END_FUNCTION_BLOCK

// ---- Observer Pattern/Abstraction/FB_AbstractObservable.TcPOU
FUNCTION_BLOCK ABSTRACT FB_AbstractObservable EXTENDS FB_Object IMPLEMENTS I_Observable
VAR
    // Attributes
    _nTypeClass:                __SYSTEM.TYPE_CLASS;
    _bAutoNotify:               BOOL := TRUE; // Notify automatically on write access of observable value
    _bNotifyWhenChanged:        BOOL; // Notify only when the value is actually changed

    // Dynamic mem
    _fbObsList:                 FB_List(0); // Observer list

    _fbNotifyObservers:         FB_NotifyObserverAction;
END_VAR

METHOD Attach : BOOL
VAR_INPUT
    ipObserver:     I_Observer;
END_VAR
IF ipObserver = 0 // Invalid interface pointer
    OR_ELSE ipObserver.nTypeClass <> THIS^._nTypeClass // Invalid type
    OR_ELSE THIS^.Contains(ipObserver) // Already added
    THEN
    RETURN;
END_IF

Attach := THIS^._fbObsList.AddItem(ipObserver) <> -1;

IF Attach THEN
    THIS^.NotifyLast();
END_IF
END_METHOD

(*Notify automatically on write access of observable value*)
PROPERTY bAutoNotify : BOOL
GET
bAutoNotify := THIS^._bAutoNotify;
END_GET
SET
THIS^._bAutoNotify := bAutoNotify;
END_SET
END_PROPERTY

PROPERTY bNotifyWhenChanged : BOOL
GET
bNotifyWhenChanged := THIS^._bNotifyWhenChanged;
END_GET
SET
THIS^._bNotifyWhenChanged := bNotifyWhenChanged;
END_SET
END_PROPERTY

METHOD ClearAll
VAR_INPUT
END_VAR
THIS^._fbObsList.Clear();
END_METHOD

METHOD Contains : BOOL
VAR_INPUT
    ipObserver: I_Observer;
END_VAR
Contains := THIS^._fbObsList.Contains(ipObserver);
END_METHOD

METHOD Detach : BOOL
VAR_INPUT
    ipObserver:     I_Observer;
END_VAR
Detach := THIS^._fbObsList.Remove(ipObserver);
END_METHOD

PROPERTY ABSTRACT nDataSize : UDINT
GET
END_GET
END_PROPERTY

PROPERTY nObserverCount : UDINT
GET
nObserverCount := THIS^._fbObsList.nCount;
END_GET
END_PROPERTY

METHOD NotifyAll : I_Observable
NotifyAll := THIS^;

THIS^._fbObsList.ForEach(
    THIS^._fbNotifyObservers
         .Inputs(THIS^.pData,
                 THIS^._nTypeClass,
                 THIS^.nDataSize));
END_METHOD

METHOD NotifyLast : I_Observable
VAR
    ipLastObs: I_Observer;
END_VAR
NotifyLast := THIS^;

ipLastObs := THIS^.ObserverAt(TO_DINT(THIS^.nObserverCount) - 1);

IF ipLastObs <> 0 THEN
    ipLastObs.UpdateP(pData := THIS^.pData,
                      nTypeClass := THIS^._nTypeClass,
                      nSize := THIS^.nDataSize);
END_IF
END_METHOD

METHOD PROTECTED NotifyWithConditions : I_Observable
VAR_INPUT
END_VAR
NotifyWithConditions := THIS^;

IF NOT THIS^._bAutoNotify THEN
    RETURN;
END_IF

IF THIS^._bNotifyWhenChanged
    AND_THEN NOT THIS^.ValueChanged() THEN
    RETURN;
END_IF

THIS^.NotifyAll();
END_METHOD

PROPERTY nTypeClass : __SYSTEM.TYPE_CLASS
GET
nTypeClass := THIS^._nTypeClass;
END_GET
END_PROPERTY

METHOD ObserverAt : I_Observer
VAR_INPUT
    nIdx: DINT;
END_VAR
__QUERYINTERFACE(THIS^._fbObsList.ItemAt(nIdx), ObserverAt);
END_METHOD

PROPERTY PROTECTED ABSTRACT pData : POINTER TO BYTE
GET
END_GET
END_PROPERTY

METHOD ABSTRACT ValueChanged : BOOL
VAR_INPUT
END_VAR
END_METHOD

END_FUNCTION_BLOCK

// ---- Observer Pattern/Abstraction/Actions/FB_NotifyObserverAction.TcPOU
FUNCTION_BLOCK FB_NotifyObserverAction EXTENDS FB_Action
VAR
    _pData: POINTER TO BYTE;
    _nSize: UDINT;
    _nTypeClass: __SYSTEM.TYPE_CLASS;
END_VAR

METHOD  Execute
VAR_INPUT
    ipObject: I_Object;
END_VAR
VAR
    ipObs: I_Observer;
END_VAR
__QUERYINTERFACE(ipObject, ipObs);

IF ipObs = 0 THEN
    RETURN;
END_IF

ipObs.UpdateP(pData := THIS^._pData,
              nTypeClass := THIS^._nTypeClass,
              nSize := THIS^._nSize);
END_METHOD

METHOD Inputs : I_Action
VAR_INPUT
    pData:          POINTER TO BYTE;
    nTypeClass:     __SYSTEM.TYPE_CLASS;
    nSize:          UDINT;
END_VAR
Inputs := THIS^;

THIS^._pData := pData;
THIS^._nTypeClass := nTypeClass;
THIS^._nSize := nSize;
END_METHOD

END_FUNCTION_BLOCK

// ---- Observer Pattern/FB_Observer_REAL.TcPOU
FUNCTION_BLOCK FB_Observer_REAL EXTENDS FB_AbstractObserver
VAR
    _fVal:              REAL;
END_VAR

METHOD FB_init : BOOL
VAR_INPUT
	bInitRetains : BOOL; // if TRUE, the retain variables are initialized (warm start / cold start)
	bInCopyCode : BOOL;  // if TRUE, the instance afterwards gets moved into the copy code (online change)
END_VAR
THIS^._nTypeClass := __SYSTEM.TYPE_CLASS.TYPE_REAL;
THIS^._pVal := ADR(THIS^._fVal);
THIS^._nSize := SIZEOF(THIS^._fVal);
END_METHOD

PROPERTY fValue32 : REAL
GET
fValue32 := THIS^._fVal;
END_GET
END_PROPERTY

END_FUNCTION_BLOCK

// ---- Observer Pattern/Abstraction/FB_AbstractObserver.TcPOU
FUNCTION_BLOCK ABSTRACT FB_AbstractObserver EXTENDS FB_Object IMPLEMENTS I_Observer
VAR
    _nTypeClass:        __SYSTEM.TYPE_CLASS;
    _pVal:              POINTER TO BYTE;
    _nSize:             DINT;
    _nUpdateCounter:    UDINT;
END_VAR

METHOD PROTECTED _Update
VAR_INPUT
    pData:          POINTER TO BYTE;
    nTypeClass:     __SYSTEM.TYPE_CLASS;
    nSize:          UDINT;
END_VAR
VAR
    nMemcpyRes:     UDINT;
END_VAR
IF nTypeClass <> THIS^._nTypeClass THEN
    RETURN;
END_IF

IF nSize <> TO_UDINT(THIS^._nSize) THEN
    RETURN;
END_IF

IF pData = 0 THEN
    RETURN;
END_IF

nMemcpyRes := Tc2_System.MEMCPY(destAddr := THIS^._pVal,
                                srcAddr := pData,
                                n := TO_UDINT(THIS^._nSize));

IF nMemcpyRes <> 0 THEN
    THIS^._nUpdateCounter := THIS^._nUpdateCounter + 1;
END_IF
END_METHOD

PROPERTY nTypeClass : __SYSTEM.TYPE_CLASS
GET
nTypeClass := THIS^._nTypeClass;
END_GET
END_PROPERTY

METHOD PROTECTED PostUpdate
VAR_INPUT
END_VAR
END_METHOD

METHOD PROTECTED PreUpdate
VAR_INPUT
END_VAR
END_METHOD

{attribute 'hasanytype'}
METHOD FINAL Update
(* Template method for updating using ANY-typed variable *)
VAR_INPUT
    anyVal:         ANY;
END_VAR
THIS^.PreUpdate();

THIS^._Update(pData := anyVal.pValue,
              nTypeClass := anyVal.TypeClass,
              nSize := TO_UDINT(anyVal.diSize));

THIS^.PostUpdate();
END_METHOD

METHOD FINAL UpdateP
(* Template method for updating using explicit
   variable information *)
VAR_INPUT
    pData:          POINTER TO BYTE;
    nTypeClass:     __SYSTEM.TYPE_CLASS;
    nSize:          UDINT;
END_VAR
THIS^.PreUpdate();

THIS^._Update(pData := pData,
              nTypeClass := nTypeClass,
              nSize := nSize);

THIS^.PostUpdate();
END_METHOD

END_FUNCTION_BLOCK

// ---- Observer Pattern/FB_Observable_DINT.TcPOU
FUNCTION_BLOCK FB_Observable_DINT EXTENDS FB_AbstractObservable
VAR
    _nVal:              DINT;
    _nOldVal:           DINT;
END_VAR

METHOD FB_init : BOOL
VAR_INPUT
    bInitRetains:       BOOL; // if TRUE, the retain variables are initialized (warm start / cold start)
    bInCopyCode:        BOOL;  // if TRUE, the instance afterwards gets moved into the copy code (online change)
END_VAR
THIS^._nTypeClass := __SYSTEM.TYPE_CLASS.TYPE_DINT;
END_METHOD

PROPERTY nDataSize : UDINT
GET
nDataSize := SIZEOF(DINT);
END_GET
END_PROPERTY

PROPERTY nValue32 : DINT
GET
nValue32 := THIS^._nVal;
END_GET
SET
THIS^._nOldVal := THIS^._nVal;
THIS^._nVal := nValue32;

THIS^.NotifyWithConditions();
END_SET
END_PROPERTY

PROPERTY PROTECTED pData : POINTER TO BYTE
GET
pData := ADR(THIS^._nVal);
END_GET
END_PROPERTY

METHOD  ValueChanged : BOOL
VAR_INPUT
END_VAR
ValueChanged := THIS^._nOldVal <> THIS^._nVal;
END_METHOD

END_FUNCTION_BLOCK

// ---- Observer Pattern/FB_Observable_UDINT.TcPOU
FUNCTION_BLOCK FB_Observable_UDINT EXTENDS FB_AbstractObservable
VAR
    _nVal:              UDINT;
    _nOldVal:           UDINT;
END_VAR

METHOD FB_init : BOOL
VAR_INPUT
    bInitRetains:       BOOL; // if TRUE, the retain variables are initialized (warm start / cold start)
    bInCopyCode:        BOOL;  // if TRUE, the instance afterwards gets moved into the copy code (online change)
END_VAR
THIS^._nTypeClass := __SYSTEM.TYPE_CLASS.TYPE_UDINT;
END_METHOD

PROPERTY nDataSize : UDINT
GET
nDataSize := SIZEOF(UDINT);
END_GET
END_PROPERTY

PROPERTY nValue32 : UDINT
GET
nValue32 := THIS^._nVal;
END_GET
SET
THIS^._nOldVal := THIS^._nVal;
THIS^._nVal := nValue32;

THIS^.NotifyWithConditions();
END_SET
END_PROPERTY

PROPERTY PROTECTED pData : POINTER TO BYTE
GET
pData := ADR(THIS^._nVal);
END_GET
END_PROPERTY

METHOD  ValueChanged : BOOL
VAR_INPUT
END_VAR
ValueChanged := THIS^._nOldVal <> THIS^._nVal;
END_METHOD

END_FUNCTION_BLOCK

// ---- Observer Pattern/FB_Observable_UINT.TcPOU
FUNCTION_BLOCK FB_Observable_UINT EXTENDS FB_AbstractObservable
VAR
    _nVal:              UINT;
    _nOldVal:           UINT;
END_VAR

METHOD FB_init : BOOL
VAR_INPUT
    bInitRetains:       BOOL; // if TRUE, the retain variables are initialized (warm start / cold start)
    bInCopyCode:        BOOL;  // if TRUE, the instance afterwards gets moved into the copy code (online change)
END_VAR
THIS^._nTypeClass := __SYSTEM.TYPE_CLASS.TYPE_UINT;
END_METHOD

PROPERTY nDataSize : UDINT
GET
nDataSize := SIZEOF(UINT);
END_GET
END_PROPERTY

PROPERTY nValue16 : UINT
GET
nValue16 := THIS^._nVal;
END_GET
SET
THIS^._nOldVal := THIS^._nVal;
THIS^._nVal := nValue16;

THIS^.NotifyWithConditions();
END_SET
END_PROPERTY

PROPERTY PROTECTED pData : POINTER TO BYTE
GET
pData := ADR(THIS^._nVal);
END_GET
END_PROPERTY

METHOD  ValueChanged : BOOL
VAR_INPUT
END_VAR
ValueChanged := THIS^._nOldVal <> THIS^._nVal;
END_METHOD

END_FUNCTION_BLOCK

// ---- Observer Pattern/FB_Observable_LREAL.TcPOU
FUNCTION_BLOCK FB_Observable_LREAL EXTENDS FB_AbstractObservable
VAR
    _fVal:                  LREAL;
    _fOldVal:               LREAL;
END_VAR

METHOD FB_init : BOOL
VAR_INPUT
    bInitRetains:       BOOL; // if TRUE, the retain variables are initialized (warm start / cold start)
    bInCopyCode:        BOOL;  // if TRUE, the instance afterwards gets moved into the copy code (online change)
END_VAR
THIS^._nTypeClass := __SYSTEM.TYPE_CLASS.TYPE_LREAL;
END_METHOD

PROPERTY fValue64 : LREAL
GET
fValue64 := THIS^._fVal;
END_GET
SET
THIS^._fOldVal := _fVal;
THIS^._fVal := fValue64;

THIS^.NotifyWithConditions();
END_SET
END_PROPERTY

PROPERTY nDataSize : UDINT
GET
nDataSize := SIZEOF(LREAL);
END_GET
END_PROPERTY

PROPERTY PROTECTED pData : POINTER TO BYTE
GET
pData := ADR(THIS^._fVal);
END_GET
END_PROPERTY

METHOD  ValueChanged : BOOL
VAR_INPUT
END_VAR
ValueChanged := THIS^._fOldVal <> THIS^._fVal;
END_METHOD

END_FUNCTION_BLOCK

// ---- Observer Pattern/FB_Observer_DINT.TcPOU
FUNCTION_BLOCK FB_Observer_DINT EXTENDS FB_AbstractObserver
VAR
    _nVal:              DINT;
END_VAR

METHOD FB_init : BOOL
VAR_INPUT
	bInitRetains : BOOL; // if TRUE, the retain variables are initialized (warm start / cold start)
	bInCopyCode : BOOL;  // if TRUE, the instance afterwards gets moved into the copy code (online change)
END_VAR
THIS^._nTypeClass := __SYSTEM.TYPE_CLASS.TYPE_DINT;
THIS^._pVal := ADR(THIS^._nVal);
THIS^._nSize := SIZEOF(THIS^._nVal);
END_METHOD

PROPERTY nValue32 : DINT
GET
nValue32 := THIS^._nVal;
END_GET
END_PROPERTY

END_FUNCTION_BLOCK

// ---- Observer Pattern/FB_Observer_UDINT.TcPOU
FUNCTION_BLOCK FB_Observer_UDINT EXTENDS FB_AbstractObserver
VAR
    _nVal:              UDINT;
END_VAR

METHOD FB_init : BOOL
VAR_INPUT
	bInitRetains : BOOL; // if TRUE, the retain variables are initialized (warm start / cold start)
	bInCopyCode : BOOL;  // if TRUE, the instance afterwards gets moved into the copy code (online change)
END_VAR
THIS^._nTypeClass := __SYSTEM.TYPE_CLASS.TYPE_UDINT;
THIS^._pVal := ADR(THIS^._nVal);
THIS^._nSize := SIZEOF(THIS^._nVal);
END_METHOD

PROPERTY nValue32 : UDINT
GET
nValue32 := THIS^._nVal;
END_GET
END_PROPERTY

END_FUNCTION_BLOCK

// ---- Observer Pattern/FB_Observer_UINT.TcPOU
FUNCTION_BLOCK FB_Observer_UINT EXTENDS FB_AbstractObserver
VAR
    _nVal:              UINT;
END_VAR

METHOD FB_init : BOOL
VAR_INPUT
	bInitRetains : BOOL; // if TRUE, the retain variables are initialized (warm start / cold start)
	bInCopyCode : BOOL;  // if TRUE, the instance afterwards gets moved into the copy code (online change)
END_VAR
THIS^._nTypeClass := __SYSTEM.TYPE_CLASS.TYPE_UINT;
THIS^._pVal := ADR(THIS^._nVal);
THIS^._nSize := SIZEOF(THIS^._nVal);
END_METHOD

PROPERTY nValue16 : UINT
GET
nValue16 := THIS^._nVal;
END_GET
END_PROPERTY

END_FUNCTION_BLOCK

// ---- Observer Pattern/FB_Observer_LREAL.TcPOU
FUNCTION_BLOCK FB_Observer_LREAL EXTENDS FB_AbstractObserver
VAR
    _fVal:              LREAL;
END_VAR

METHOD FB_init : BOOL
VAR_INPUT
	bInitRetains : BOOL; // if TRUE, the retain variables are initialized (warm start / cold start)
	bInCopyCode : BOOL;  // if TRUE, the instance afterwards gets moved into the copy code (online change)
END_VAR
THIS^._nTypeClass := __SYSTEM.TYPE_CLASS.TYPE_LREAL;
THIS^._pVal := ADR(THIS^._fVal);
THIS^._nSize := SIZEOF(THIS^._fVal);
END_METHOD

PROPERTY fValue64 : LREAL
GET
fValue64 := THIS^._fVal;
END_GET
END_PROPERTY

END_FUNCTION_BLOCK

// ---- Observer Pattern/FB_Observable_BOOL.TcPOU
FUNCTION_BLOCK FB_Observable_BOOL EXTENDS FB_AbstractObservable
VAR
    _bVal:      BOOL;
    _bOldVal:   BOOL;
END_VAR

PROPERTY PUBLIC bVal : BOOL
GET
bVal := THIS^._bVal;
END_GET
SET
THIS^._bOldVal := THIS^._bVal;
THIS^._bVal := bVal;

THIS^.NotifyWithConditions();
END_SET
END_PROPERTY

METHOD FB_init : BOOL
VAR_INPUT
    bInitRetains:       BOOL; // if TRUE, the retain variables are initialized (warm start / cold start)
    bInCopyCode:        BOOL;  // if TRUE, the instance afterwards gets moved into the copy code (online change)
END_VAR
THIS^._nTypeClass := __SYSTEM.TYPE_CLASS.TYPE_BOOL;
END_METHOD

PROPERTY nDataSize : UDINT
GET
nDataSize := SIZEOF(BOOL);
END_GET
END_PROPERTY

PROPERTY PROTECTED pData : POINTER TO BYTE
GET
pData := ADR(THIS^._bVal);
END_GET
END_PROPERTY

METHOD  ValueChanged : BOOL
VAR_INPUT
END_VAR
ValueChanged := THIS^._bOldVal <> THIS^._bVal;
END_METHOD

END_FUNCTION_BLOCK

// ---- Observer Pattern/FB_Observable_BYTE.TcPOU
FUNCTION_BLOCK FB_Observable_BYTE EXTENDS FB_AbstractObservable
VAR
    _nVal:              BYTE;
    _nOldVal:           BYTE;
END_VAR

METHOD FB_init : BOOL
VAR_INPUT
    bInitRetains:       BOOL; // if TRUE, the retain variables are initialized (warm start / cold start)
    bInCopyCode:        BOOL;  // if TRUE, the instance afterwards gets moved into the copy code (online change)
END_VAR
THIS^._nTypeClass := __SYSTEM.TYPE_CLASS.TYPE_BYTE;
END_METHOD

PROPERTY nDataSize : UDINT
GET
nDataSize := SIZEOF(BYTE);
END_GET
END_PROPERTY

PROPERTY nValue8 : BYTE
GET
nValue8 := THIS^._nVal;
END_GET
SET
THIS^._nOldVal := THIS^._nVal;
THIS^._nVal := nValue8;

THIS^.NotifyWithConditions();
END_SET
END_PROPERTY

PROPERTY PROTECTED pData : POINTER TO BYTE
GET
pData := ADR(THIS^._nVal);
END_GET
END_PROPERTY

METHOD  ValueChanged : BOOL
VAR_INPUT
END_VAR
ValueChanged := THIS^._nOldVal <> THIS^._nVal;
END_METHOD

END_FUNCTION_BLOCK

// ---- Observer Pattern/FB_Observable_WORD.TcPOU
FUNCTION_BLOCK FB_Observable_WORD EXTENDS FB_AbstractObservable
VAR
    _nVal:              WORD;
    _nOldVal:           WORD;
END_VAR

METHOD FB_init : BOOL
VAR_INPUT
    bInitRetains:       BOOL; // if TRUE, the retain variables are initialized (warm start / cold start)
    bInCopyCode:        BOOL;  // if TRUE, the instance afterwards gets moved into the copy code (online change)
END_VAR
THIS^._nTypeClass := __SYSTEM.TYPE_CLASS.TYPE_WORD;
END_METHOD

PROPERTY nDataSize : UDINT
GET
nDataSize := SIZEOF(WORD);
END_GET
END_PROPERTY

PROPERTY nValue16 : WORD
GET
nValue16 := THIS^._nVal;
END_GET
SET
THIS^._nOldVal := THIS^._nVal;
THIS^._nVal := nValue16;

THIS^.NotifyWithConditions();
END_SET
END_PROPERTY

PROPERTY PROTECTED pData : POINTER TO BYTE
GET
pData := ADR(THIS^._nVal);
END_GET
END_PROPERTY

METHOD  ValueChanged : BOOL
VAR_INPUT
END_VAR
ValueChanged := THIS^._nOldVal <> THIS^._nVal;
END_METHOD

END_FUNCTION_BLOCK

// ---- Observer Pattern/FB_Observable_DWORD.TcPOU
FUNCTION_BLOCK FB_Observable_DWORD EXTENDS FB_AbstractObservable
VAR
    _nVal:              DWORD;
    _nOldVal:           DWORD;
END_VAR

METHOD FB_init : BOOL
VAR_INPUT
    bInitRetains:       BOOL; // if TRUE, the retain variables are initialized (warm start / cold start)
    bInCopyCode:        BOOL;  // if TRUE, the instance afterwards gets moved into the copy code (online change)
END_VAR
THIS^._nTypeClass := __SYSTEM.TYPE_CLASS.TYPE_DWORD;
END_METHOD

PROPERTY nDataSize : UDINT
GET
nDataSize := SIZEOF(DWORD);
END_GET
END_PROPERTY

PROPERTY nValue32 : DWORD
GET
nValue32 := THIS^._nVal;
END_GET
SET
THIS^._nOldVal := THIS^._nVal;
THIS^._nVal := nValue32;

THIS^.NotifyWithConditions();
END_SET
END_PROPERTY

PROPERTY PROTECTED pData : POINTER TO BYTE
GET
pData := ADR(THIS^._nVal);
END_GET
END_PROPERTY

METHOD  ValueChanged : BOOL
VAR_INPUT
END_VAR
ValueChanged := THIS^._nOldVal <> THIS^._nVal;
END_METHOD

END_FUNCTION_BLOCK

// ---- Observer Pattern/FB_Observable_LWORD.TcPOU
FUNCTION_BLOCK FB_Observable_LWORD EXTENDS FB_AbstractObservable
VAR
    _nVal:              LWORD;
    _nOldVal:           LWORD;
END_VAR

METHOD FB_init : BOOL
VAR_INPUT
    bInitRetains:       BOOL; // if TRUE, the retain variables are initialized (warm start / cold start)
    bInCopyCode:        BOOL;  // if TRUE, the instance afterwards gets moved into the copy code (online change)
END_VAR
THIS^._nTypeClass := __SYSTEM.TYPE_CLASS.TYPE_LWORD;
END_METHOD

PROPERTY nDataSize : UDINT
GET
nDataSize := SIZEOF(LWORD);
END_GET
END_PROPERTY

PROPERTY nValue64 : LWORD
GET
nValue64 := THIS^._nVal;
END_GET
SET
THIS^._nOldVal := THIS^._nVal;
THIS^._nVal := nValue64;

THIS^.NotifyWithConditions();
END_SET
END_PROPERTY

PROPERTY PROTECTED pData : POINTER TO BYTE
GET
pData := ADR(THIS^._nVal);
END_GET
END_PROPERTY

METHOD  ValueChanged : BOOL
VAR_INPUT
END_VAR
ValueChanged := THIS^._nOldVal <> THIS^._nVal;
END_METHOD

END_FUNCTION_BLOCK

// ---- Observer Pattern/FB_Observable_SINT.TcPOU
FUNCTION_BLOCK FB_Observable_SINT EXTENDS FB_AbstractObservable
VAR
    _nVal:              SINT;
    _nOldVal:           SINT;
END_VAR

METHOD FB_init : BOOL
VAR_INPUT
    bInitRetains:       BOOL; // if TRUE, the retain variables are initialized (warm start / cold start)
    bInCopyCode:        BOOL;  // if TRUE, the instance afterwards gets moved into the copy code (online change)
END_VAR
THIS^._nTypeClass := __SYSTEM.TYPE_CLASS.TYPE_SINT;
END_METHOD

PROPERTY nDataSize : UDINT
GET
nDataSize := SIZEOF(SINT);
END_GET
END_PROPERTY

PROPERTY nValue8 : SINT
GET
nValue8 := THIS^._nVal;
END_GET
SET
THIS^._nOldVal := THIS^._nVal;
THIS^._nVal := nValue8;

THIS^.NotifyWithConditions();
END_SET
END_PROPERTY

PROPERTY PROTECTED pData : POINTER TO BYTE
GET
pData := ADR(THIS^._nVal);
END_GET
END_PROPERTY

METHOD  ValueChanged : BOOL
VAR_INPUT
END_VAR
ValueChanged := THIS^._nOldVal <> THIS^._nVal;
END_METHOD

END_FUNCTION_BLOCK

// ---- Observer Pattern/FB_Observable_USINT.TcPOU
FUNCTION_BLOCK FB_Observable_USINT EXTENDS FB_AbstractObservable
VAR
    _nVal:              USINT;
    _nOldVal:           USINT;
END_VAR

METHOD FB_init : BOOL
VAR_INPUT
    bInitRetains:       BOOL; // if TRUE, the retain variables are initialized (warm start / cold start)
    bInCopyCode:        BOOL;  // if TRUE, the instance afterwards gets moved into the copy code (online change)
END_VAR
THIS^._nTypeClass := __SYSTEM.TYPE_CLASS.TYPE_USINT;
END_METHOD

PROPERTY nDataSize : UDINT
GET
nDataSize := SIZEOF(USINT);
END_GET
END_PROPERTY

PROPERTY nValue8 : USINT
GET
nValue8 := THIS^._nVal;
END_GET
SET
THIS^._nOldVal := THIS^._nVal;
THIS^._nVal := nValue8;

THIS^.NotifyWithConditions();
END_SET
END_PROPERTY

PROPERTY PROTECTED pData : POINTER TO BYTE
GET
pData := ADR(THIS^._nVal);
END_GET
END_PROPERTY

METHOD  ValueChanged : BOOL
VAR_INPUT
END_VAR
ValueChanged := THIS^._nOldVal <> THIS^._nVal;
END_METHOD

END_FUNCTION_BLOCK

// ---- Observer Pattern/FB_Observable_INT.TcPOU
FUNCTION_BLOCK FB_Observable_INT EXTENDS FB_AbstractObservable
VAR
    _nVal:              INT;
    _nOldVal:           INT;
END_VAR

METHOD FB_init : BOOL
VAR_INPUT
    bInitRetains:       BOOL; // if TRUE, the retain variables are initialized (warm start / cold start)
    bInCopyCode:        BOOL;  // if TRUE, the instance afterwards gets moved into the copy code (online change)
END_VAR
THIS^._nTypeClass := __SYSTEM.TYPE_CLASS.TYPE_INT;
END_METHOD

PROPERTY nDataSize : UDINT
GET
nDataSize := SIZEOF(INT);
END_GET
END_PROPERTY

PROPERTY nValue16 : INT
GET
nValue16 := THIS^._nVal;
END_GET
SET
THIS^._nOldVal := THIS^._nVal;
THIS^._nVal := nValue16;

THIS^.NotifyWithConditions();
END_SET
END_PROPERTY

PROPERTY PROTECTED pData : POINTER TO BYTE
GET
pData := ADR(THIS^._nVal);
END_GET
END_PROPERTY

METHOD  ValueChanged : BOOL
VAR_INPUT
END_VAR
ValueChanged := THIS^._nOldVal <> THIS^._nVal;
END_METHOD

END_FUNCTION_BLOCK

// ---- Observer Pattern/FB_Observable_LINT.TcPOU
FUNCTION_BLOCK FB_Observable_LINT EXTENDS FB_AbstractObservable
VAR
    _nVal:              LINT;
    _nOldVal:           LINT;
END_VAR

METHOD FB_init : BOOL
VAR_INPUT
    bInitRetains:       BOOL; // if TRUE, the retain variables are initialized (warm start / cold start)
    bInCopyCode:        BOOL;  // if TRUE, the instance afterwards gets moved into the copy code (online change)
END_VAR
THIS^._nTypeClass := __SYSTEM.TYPE_CLASS.TYPE_LINT;
END_METHOD

PROPERTY nDataSize : UDINT
GET
nDataSize := SIZEOF(LINT);
END_GET
END_PROPERTY

PROPERTY nValue64 : LINT
GET
nValue64 := THIS^._nVal;
END_GET
SET
THIS^._nOldVal := THIS^._nVal;
THIS^._nVal := nValue64;

THIS^.NotifyWithConditions();
END_SET
END_PROPERTY

PROPERTY PROTECTED pData : POINTER TO BYTE
GET
pData := ADR(THIS^._nVal);
END_GET
END_PROPERTY

METHOD  ValueChanged : BOOL
VAR_INPUT
END_VAR
ValueChanged := THIS^._nOldVal <> THIS^._nVal;
END_METHOD

END_FUNCTION_BLOCK

// ---- Observer Pattern/FB_Observable_ULINT.TcPOU
FUNCTION_BLOCK FB_Observable_ULINT EXTENDS FB_AbstractObservable
VAR
    _nVal:              ULINT;
    _nOldVal:           ULINT;
END_VAR

METHOD FB_init : BOOL
VAR_INPUT
    bInitRetains:       BOOL; // if TRUE, the retain variables are initialized (warm start / cold start)
    bInCopyCode:        BOOL;  // if TRUE, the instance afterwards gets moved into the copy code (online change)
END_VAR
THIS^._nTypeClass := __SYSTEM.TYPE_CLASS.TYPE_ULINT;
END_METHOD

PROPERTY nDataSize : UDINT
GET
nDataSize := SIZEOF(LINT);
END_GET
END_PROPERTY

PROPERTY nValue64 : ULINT
GET
nValue64 := THIS^._nVal;
END_GET
SET
THIS^._nOldVal := THIS^._nVal;
THIS^._nVal := nValue64;

THIS^.NotifyWithConditions();
END_SET
END_PROPERTY

PROPERTY PROTECTED pData : POINTER TO BYTE
GET
pData := ADR(THIS^._nVal);
END_GET
END_PROPERTY

METHOD  ValueChanged : BOOL
VAR_INPUT
END_VAR
ValueChanged := THIS^._nOldVal <> THIS^._nVal;
END_METHOD

END_FUNCTION_BLOCK

// ---- Observer Pattern/FB_Observer_BOOL.TcPOU
FUNCTION_BLOCK FB_Observer_BOOL EXTENDS FB_AbstractObserver
VAR
    _bVal:      BOOL;
END_VAR

PROPERTY bValue : BOOL
GET
bValue := THIS^._bVal;
END_GET
END_PROPERTY

METHOD FB_init : BOOL
VAR_INPUT
	bInitRetains : BOOL; // if TRUE, the retain variables are initialized (warm start / cold start)
	bInCopyCode : BOOL;  // if TRUE, the instance afterwards gets moved into the copy code (online change)
END_VAR
THIS^._nTypeClass := __SYSTEM.TYPE_CLASS.TYPE_BOOL;
THIS^._pVal := ADR(THIS^._bVal);
THIS^._nSize := SIZEOF(THIS^._bVal);
END_METHOD

END_FUNCTION_BLOCK

// ---- Observer Pattern/FB_Observer_BYTE.TcPOU
FUNCTION_BLOCK FB_Observer_BYTE EXTENDS FB_AbstractObserver
VAR
    _nVal:              BYTE;
END_VAR

METHOD FB_init : BOOL
VAR_INPUT
	bInitRetains : BOOL; // if TRUE, the retain variables are initialized (warm start / cold start)
	bInCopyCode : BOOL;  // if TRUE, the instance afterwards gets moved into the copy code (online change)
END_VAR
THIS^._nTypeClass := __SYSTEM.TYPE_CLASS.TYPE_BYTE;
THIS^._pVal := ADR(THIS^._nVal);
THIS^._nSize := SIZEOF(THIS^._nVal);
END_METHOD

PROPERTY nValue8 : BYTE
GET
nValue8 := THIS^._nVal;
END_GET
END_PROPERTY

END_FUNCTION_BLOCK

// ---- Observer Pattern/FB_Observer_WORD.TcPOU
FUNCTION_BLOCK FB_Observer_WORD EXTENDS FB_AbstractObserver
VAR
    _nVal:              WORD;
END_VAR

METHOD FB_init : BOOL
VAR_INPUT
	bInitRetains : BOOL; // if TRUE, the retain variables are initialized (warm start / cold start)
	bInCopyCode : BOOL;  // if TRUE, the instance afterwards gets moved into the copy code (online change)
END_VAR
THIS^._nTypeClass := __SYSTEM.TYPE_CLASS.TYPE_WORD;
THIS^._pVal := ADR(THIS^._nVal);
THIS^._nSize := SIZEOF(THIS^._nVal);
END_METHOD

PROPERTY nValue16 : WORD
GET
nValue16 := THIS^._nVal;
END_GET
END_PROPERTY

END_FUNCTION_BLOCK

// ---- Observer Pattern/FB_Observer_DWORD.TcPOU
FUNCTION_BLOCK FB_Observer_DWORD EXTENDS FB_AbstractObserver
VAR
    _nVal:              DWORD;
END_VAR

METHOD FB_init : BOOL
VAR_INPUT
	bInitRetains : BOOL; // if TRUE, the retain variables are initialized (warm start / cold start)
	bInCopyCode : BOOL;  // if TRUE, the instance afterwards gets moved into the copy code (online change)
END_VAR
THIS^._nTypeClass := __SYSTEM.TYPE_CLASS.TYPE_DWORD;
THIS^._pVal := ADR(THIS^._nVal);
THIS^._nSize := SIZEOF(THIS^._nVal);
END_METHOD

PROPERTY nValue32 : DWORD
GET
nValue32 := THIS^._nVal;
END_GET
END_PROPERTY

END_FUNCTION_BLOCK

// ---- Observer Pattern/FB_Observer_LWORD.TcPOU
FUNCTION_BLOCK FB_Observer_LWORD EXTENDS FB_AbstractObserver
VAR
    _nVal:              LWORD;
END_VAR

METHOD FB_init : BOOL
VAR_INPUT
	bInitRetains : BOOL; // if TRUE, the retain variables are initialized (warm start / cold start)
	bInCopyCode : BOOL;  // if TRUE, the instance afterwards gets moved into the copy code (online change)
END_VAR
THIS^._nTypeClass := __SYSTEM.TYPE_CLASS.TYPE_LWORD;
THIS^._pVal := ADR(THIS^._nVal);
THIS^._nSize := SIZEOF(THIS^._nVal);
END_METHOD

PROPERTY nValue64 : LWORD
GET
nValue64 := THIS^._nVal;
END_GET
END_PROPERTY

END_FUNCTION_BLOCK

// ---- Observer Pattern/FB_Observer_SINT.TcPOU
FUNCTION_BLOCK FB_Observer_SINT EXTENDS FB_AbstractObserver
VAR
    _nVal:              SINT;
END_VAR

METHOD FB_init : BOOL
VAR_INPUT
	bInitRetains : BOOL; // if TRUE, the retain variables are initialized (warm start / cold start)
	bInCopyCode : BOOL;  // if TRUE, the instance afterwards gets moved into the copy code (online change)
END_VAR
THIS^._nTypeClass := __SYSTEM.TYPE_CLASS.TYPE_SINT;
THIS^._pVal := ADR(THIS^._nVal);
THIS^._nSize := SIZEOF(THIS^._nVal);
END_METHOD

PROPERTY nValue8 : SINT
GET
nValue8 := THIS^._nVal;
END_GET
END_PROPERTY

END_FUNCTION_BLOCK

// ---- Observer Pattern/FB_Observer_USINT.TcPOU
FUNCTION_BLOCK FB_Observer_USINT EXTENDS FB_AbstractObserver
VAR
    _nVal:              USINT;
END_VAR

METHOD FB_init : BOOL
VAR_INPUT
	bInitRetains : BOOL; // if TRUE, the retain variables are initialized (warm start / cold start)
	bInCopyCode : BOOL;  // if TRUE, the instance afterwards gets moved into the copy code (online change)
END_VAR
THIS^._nTypeClass := __SYSTEM.TYPE_CLASS.TYPE_USINT;
THIS^._pVal := ADR(THIS^._nVal);
THIS^._nSize := SIZEOF(THIS^._nVal);
END_METHOD

PROPERTY nValue8 : USINT
GET
nValue8 := THIS^._nVal;
END_GET
END_PROPERTY

END_FUNCTION_BLOCK

// ---- Observer Pattern/FB_Observer_INT.TcPOU
FUNCTION_BLOCK FB_Observer_INT EXTENDS FB_AbstractObserver
VAR
    _nVal:              INT;
END_VAR

METHOD FB_init : BOOL
VAR_INPUT
	bInitRetains : BOOL; // if TRUE, the retain variables are initialized (warm start / cold start)
	bInCopyCode : BOOL;  // if TRUE, the instance afterwards gets moved into the copy code (online change)
END_VAR
THIS^._nTypeClass := __SYSTEM.TYPE_CLASS.TYPE_INT;
THIS^._pVal := ADR(THIS^._nVal);
THIS^._nSize := SIZEOF(THIS^._nVal);
END_METHOD

PROPERTY nValue16 : INT
GET
nValue16 := THIS^._nVal;
END_GET
END_PROPERTY

END_FUNCTION_BLOCK

// ---- Observer Pattern/FB_Observer_LINT.TcPOU
FUNCTION_BLOCK FB_Observer_LINT EXTENDS FB_AbstractObserver
VAR
    _nVal:              LINT;
END_VAR

METHOD FB_init : BOOL
VAR_INPUT
	bInitRetains : BOOL; // if TRUE, the retain variables are initialized (warm start / cold start)
	bInCopyCode : BOOL;  // if TRUE, the instance afterwards gets moved into the copy code (online change)
END_VAR
THIS^._nTypeClass := __SYSTEM.TYPE_CLASS.TYPE_LINT;
THIS^._pVal := ADR(THIS^._nVal);
THIS^._nSize := SIZEOF(THIS^._nVal);
END_METHOD

PROPERTY nValue64 : LINT
GET
nValue64 := THIS^._nVal;
END_GET
END_PROPERTY

END_FUNCTION_BLOCK

// ---- Observer Pattern/FB_Observer_ULINT.TcPOU
FUNCTION_BLOCK FB_Observer_ULINT EXTENDS FB_AbstractObserver
VAR
    _nVal:              ULINT;
END_VAR

METHOD FB_init : BOOL
VAR_INPUT
	bInitRetains : BOOL; // if TRUE, the retain variables are initialized (warm start / cold start)
	bInCopyCode : BOOL;  // if TRUE, the instance afterwards gets moved into the copy code (online change)
END_VAR
THIS^._nTypeClass := __SYSTEM.TYPE_CLASS.TYPE_ULINT;
THIS^._pVal := ADR(THIS^._nVal);
THIS^._nSize := SIZEOF(THIS^._nVal);
END_METHOD

PROPERTY nValue64 : ULINT
GET
nValue64 := THIS^._nVal;
END_GET
END_PROPERTY

END_FUNCTION_BLOCK

// ---- Observer Pattern/FB_ObserverExt.TcPOU
FUNCTION_BLOCK FB_ObserverExt EXTENDS FB_AbstractObserver
VAR
    
END_VAR

METHOD FB_init : BOOL
VAR_INPUT
    bInitRetains: BOOL; // if TRUE, the retain variables are initialized (warm start / cold start)
    bInCopyCode: BOOL;  // if TRUE, the instance afterwards gets moved into the copy code (online change)
    anyVal: ANY;
END_VAR
THIS^._nTypeClass := anyVal.TypeClass;
THIS^._pVal := anyVal.pValue;
THIS^._nSize := anyVal.diSize;
END_METHOD

PROPERTY nSize : UDINT
GET
nSize := TO_UDINT(THIS^._nSize);
END_GET
END_PROPERTY

PROPERTY nTypeClass : __SYSTEM.TYPE_CLASS
GET
nTypeClass := THIS^._nTypeClass;
END_GET
END_PROPERTY

PROPERTY pVal : POINTER TO BYTE
GET
pVal := THIS^._pVal;
END_GET
END_PROPERTY

END_FUNCTION_BLOCK

// ---- Observer Pattern/Tests/FB_Observer_LREAL_.TcPOU
FUNCTION_BLOCK INTERNAL FB_Observer_LREAL_ EXTENDS FB_Observer_LREAL
VAR_INPUT
END_VAR
VAR_OUTPUT
END_VAR
VAR
END_VAR

PROPERTY nUpdateCounter : UDINT
GET
nUpdateCounter := THIS^._nUpdateCounter;
END_GET
END_PROPERTY

END_FUNCTION_BLOCK

// ---- State Pattern/Tests/FB_StatePattern_Test.TcPOU
FUNCTION_BLOCK INTERNAL FB_StatePattern_Test EXTENDS TcUnit.FB_TestSuite IMPLEMENTS I_Object
VAR
    _ipSelf:            I_Object;

    fbStateMachine1:    FB_StateMachine1;
    fbState11:          FB_State1(0);
    fbState12:          FB_State2(0);
    fbState13:          FB_State3(0);
    fbState14:          FB_State4(0);

    fbStateMachine2:    FB_StateMachine1;
    fbState21:          FB_State1(THIS^.fbStateMachine2);
    fbState22:          FB_State2(THIS^.fbStateMachine2);
    fbState23:          FB_State3(THIS^.fbStateMachine2);
    fbState24:          FB_State4(THIS^.fbStateMachine2);

    fbYear:             FB_Year;
END_VAR

TestAdd4StatesByInitializationExpectSuccess();
TestAdd4StatesManuallyExpectSuccess();
TestClearAllStatesExpectSuccess();
TestSeasonStateMachineAllSeasons();

METHOD Equals : BOOL
VAR_INPUT
    ipObject:       I_Object;
END_VAR
Equals := ipObject = THIS^._ipSelf;
END_METHOD

PROPERTY ipContext : I_Context
GET
ipContext := 0;
END_GET
END_PROPERTY

PROPERTY nIdentity : ULINT
GET
nIdentity := ADR(THIS^);
END_GET
END_PROPERTY

PROPERTY sPath : STRING(MAX_STRING_LENGTH)
GET
sPath := '';
END_GET
END_PROPERTY

METHOD PRIVATE TestAdd4StatesByInitializationExpectSuccess
TcUnit.TEST('TestAdd4StatesByInitializationExpectSuccess');

THIS^.AssertEquals_UDINT(Expected := 4,
                         Actual := THIS^.fbStateMachine2.nStateCount,
                         Message := 'Unexpected number of states added to state machine');
THIS^.AssertTrue(Condition := THIS^.fbStateMachine2.Contains(THIS^.fbState21),
                 Message := 'State machine does not contain added state fbState5');
THIS^.AssertTrue(Condition := THIS^.fbStateMachine2.Contains(THIS^.fbState22),
                 Message := 'State machine does not contain added state fbState6');
THIS^.AssertTrue(Condition := THIS^.fbStateMachine2.Contains(THIS^.fbState23),
                 Message := 'State machine does not contain added state fbState7');
THIS^.AssertTrue(Condition := THIS^.fbStateMachine2.Contains(THIS^.fbState24),
                 Message := 'State machine does not contain added state fbState8');

THIS^.AssertTrue(Condition := THIS^.fbState21.ipStateMachine.Equals(THIS^.fbStateMachine2),
                 Message := 'State fbState5 does not point to the correct state machine');
THIS^.AssertTrue(Condition := THIS^.fbState22.ipStateMachine.Equals(THIS^.fbStateMachine2),
                 Message := 'State fbState6 does not point to the correct state machine');
THIS^.AssertTrue(Condition := THIS^.fbState23.ipStateMachine.Equals(THIS^.fbStateMachine2),
                 Message := 'State fbState7 does not point to the correct state machine');
THIS^.AssertTrue(Condition := THIS^.fbState24.ipStateMachine.Equals(THIS^.fbStateMachine2),
                 Message := 'State fbState8 does not point to the correct state machine');


TcUnit.TEST_FINISHED();
END_METHOD

METHOD PRIVATE TestAdd4StatesManuallyExpectSuccess
TcUnit.TEST_ORDERED('TestAdd4StatesManuallyExpectSuccess');

THIS^.AssertTrue(Condition := THIS^.fbStateMachine1.AddState(THIS^.fbState11),
                 Message := 'Failed to add fbState1 to fbStateMachine');
THIS^.AssertFalse(Condition := THIS^.fbStateMachine1.AddState(THIS^.fbState11),
                  Message := 'fbState1 has already been added to fbStateMachine');
THIS^.AssertEquals_UDINT(Expected := 1,
                         Actual := THIS^.fbStateMachine1.nStateCount,
                         Message := 'Unexpected number of states added to state machine');
THIS^.AssertTrue(Condition := THIS^.fbState11.ipStateMachine.Equals(THIS^.fbStateMachine1),
                 Message := 'State fbState1 does not point to the correct state machine');

THIS^.AssertTrue(Condition := THIS^.fbStateMachine1.AddState(THIS^.fbState12),
                 Message := 'Failed to add fbState2 to fbStateMachine');
THIS^.AssertFalse(Condition := THIS^.fbStateMachine1.AddState(THIS^.fbState12),
                  Message := 'fbState2 has already been added to fbStateMachine');
THIS^.AssertEquals_UDINT(Expected := 2,
                         Actual := THIS^.fbStateMachine1.nStateCount,
                         Message := 'Unexpected number of states added to state machine');
THIS^.AssertTrue(Condition := THIS^.fbState12.ipStateMachine.Equals(THIS^.fbStateMachine1),
                 Message := 'State fbState2 does not point to the correct state machine');

THIS^.AssertTrue(Condition := THIS^.fbStateMachine1.AddState(THIS^.fbState13),
                 Message := 'Failed to add fbState3 to fbStateMachine');
THIS^.AssertFalse(Condition := THIS^.fbStateMachine1.AddState(THIS^.fbState13),
                  Message := 'fbState2 has already been added to fbStateMachine');
THIS^.AssertEquals_UDINT(Expected := 3,
                         Actual := THIS^.fbStateMachine1.nStateCount,
                         Message := 'Unexpected number of states added to state machine');
THIS^.AssertTrue(Condition := THIS^.fbState13.ipStateMachine.Equals(THIS^.fbStateMachine1),
                 Message := 'State fbState3 does not point to the correct state machine');

THIS^.AssertTrue(Condition := THIS^.fbStateMachine1.AddState(THIS^.fbState14),
                 Message := 'Failed to add fbState4 to fbStateMachine');
THIS^.AssertFalse(Condition := THIS^.fbStateMachine1.AddState(THIS^.fbState14),
                  Message := 'fbState2 has already been added to fbStateMachine');
THIS^.AssertEquals_UDINT(Expected := 4,
                         Actual := THIS^.fbStateMachine1.nStateCount,
                         Message := 'Unexpected number of states added to state machine');
THIS^.AssertTrue(Condition := THIS^.fbState14.ipStateMachine.Equals(THIS^.fbStateMachine1),
                 Message := 'State fbState4 does not point to the correct state machine');

THIS^.AssertTrue(Condition := THIS^.fbStateMachine1.Contains(THIS^.fbState11),
                 Message := 'State machine does not contain added state fbState1');
THIS^.AssertTrue(Condition := THIS^.fbStateMachine1.Contains(THIS^.fbState12),
                 Message := 'State machine does not contain added state fbState2');
THIS^.AssertTrue(Condition := THIS^.fbStateMachine1.Contains(THIS^.fbState13),
                 Message := 'State machine does not contain added state fbState3');
THIS^.AssertTrue(Condition := THIS^.fbStateMachine1.Contains(THIS^.fbState14),
                 Message := 'State machine does not contain added state fbState4');

TcUnit.TEST_FINISHED();
END_METHOD

METHOD PRIVATE TestClearAllStatesExpectSuccess
VAR_INPUT
END_VAR
TcUnit.TEST_ORDERED('TestClearAllStatesExpectSuccess');

THIS^.fbStateMachine1.ClearStates();

THIS^.AssertEquals_UDINT(Expected := 0,
                         Actual := THIS^.fbStateMachine1.nStateCount,
                         Message := 'State machine did not clear all states correctly');

THIS^.AssertFalse(Condition := THIS^.fbStateMachine1.Contains(THIS^.fbState11),
                  Message := 'Cleared state should not be in state machine');
THIS^.AssertFalse(Condition := THIS^.fbStateMachine1.Contains(THIS^.fbState12),
                  Message := 'Cleared state should not be in state machine');
THIS^.AssertFalse(Condition := THIS^.fbStateMachine1.Contains(THIS^.fbState13),
                  Message := 'Cleared state should not be in state machine');
THIS^.AssertFalse(Condition := THIS^.fbStateMachine1.Contains(THIS^.fbState14),
                  Message := 'Cleared state should not be in state machine');

TcUnit.TEST_FINISHED();
END_METHOD

METHOD PRIVATE TestSeasonStateMachineAllSeasons
VAR_INPUT
END_VAR
TcUnit.TEST('TestSeasonStateMachineAllSeasons');

THIS^.fbYear.Run();

// Summer
THIS^.AssertEquals_BYTE(Expected := 1,
                        Actual := THIS^.fbYear.CurrentState().nTyresType,
                        Message := 'Tyres initialization is incorrect for Summer');
THIS^.AssertTrue(Condition := THIS^.fbYear.CurrentState().Equals(THIS^.fbYear.StateSummer),
                 Message := 'Expected Summer to be the starting season');
THIS^.AssertTrue(Condition := THIS^.fbYear.CurrentState().bSunShining,
                 Message := 'Expected the sun to shine during Summer');
THIS^.AssertEquals_BYTE(Expected := 1,
                        Actual := THIS^.fbYear.CurrentState().nLeavesState,
                        Message := 'Expected the color of the leaves to be green');
THIS^.fbYear.ChangeToWinterTyres();
THIS^.AssertEquals_BYTE(Expected := 1,
                        Actual := THIS^.fbYear.CurrentState().nTyresType,
                        Message := 'Must not be able to put winter tyres on during Summer');

// Autumn
THIS^.fbYear.NextSeason();
THIS^.AssertTrue(Condition := THIS^.fbYear.CurrentState().Equals(THIS^.fbYear.StateAutumn),
                 Message := 'Expected Autumn to be after Summer');
THIS^.AssertTrue(Condition := THIS^.fbYear.CurrentState().bWindBlowing,
                 Message := 'Expected the wind to blow during Autumn');
THIS^.AssertEquals_BYTE(Expected := 2,
                        Actual := THIS^.fbYear.CurrentState().nLeavesState,
                        Message := 'Expected the color of the leaves to be (changing to) yellow/orange/red');
THIS^.fbYear.ChangeToWinterTyres();
THIS^.AssertEquals_BYTE(Expected := 1,
                        Actual := THIS^.fbYear.CurrentState().nTyresType,
                        Message := 'Must not be able to put winter tyres on during Autumn');

// Winter
THIS^.fbYear.NextSeason();
THIS^.AssertTrue(Condition := THIS^.fbYear.CurrentState().Equals(THIS^.fbYear.StateWinter),
                 Message := 'Expected Winter to be after Autumn');
THIS^.AssertTrue(Condition := THIS^.fbYear.CurrentState().bSnowing,
                 Message := 'Expected snow during Winter');
THIS^.AssertEquals_BYTE(Expected := 0,
                        Actual := THIS^.fbYear.CurrentState().nLeavesState,
                        Message := 'Expected (some) leaves to have been fallen off');
THIS^.fbYear.ChangeToWinterTyres();
THIS^.AssertEquals_BYTE(Expected := 0,
                        Actual := THIS^.fbYear.CurrentState().nTyresType,
                        Message := 'Failed to be able to put winter tyres on');

// Spring
THIS^.fbYear.NextSeason();
THIS^.AssertTrue(Condition := THIS^.fbYear.CurrentState().Equals(THIS^.fbYear.StateSpring),
                 Message := 'Expected Spring to be after Winter');
THIS^.AssertTrue(Condition := THIS^.fbYear.CurrentState().bRaining,
                 Message := 'Expected rain during Spring');
THIS^.AssertEquals_BYTE(Expected := 1,
                        Actual := THIS^.fbYear.CurrentState().nLeavesState,
                        Message := 'Expected the color of the leaves to be green');
THIS^.fbYear.ChangeToSummerTyres();
THIS^.AssertEquals_BYTE(Expected := 1,
                        Actual := THIS^.fbYear.CurrentState().nTyresType,
                        Message := 'Failed to be able to put summer tyres on');

TcUnit.TEST_FINISHED();
END_METHOD

END_FUNCTION_BLOCK

// ---- State Pattern/Tests/Test Subjects/FB_StateMachine1.TcPOU
FUNCTION_BLOCK INTERNAL FB_StateMachine1 EXTENDS FB_StateMachine
VAR_INPUT
END_VAR
VAR_OUTPUT
END_VAR
VAR
END_VAR

END_FUNCTION_BLOCK

// ---- State Pattern/FB_StateMachine.TcPOU
FUNCTION_BLOCK ABSTRACT FB_StateMachine EXTENDS FB_Object IMPLEMENTS I_StateMachine
VAR
    _ipState:               I_State; // Current state
    _ipPrevState:           I_State; // Previous state
    _nStateChangeCount:     UDINT := 0;
    fbStateList:            FB_List(0); // List of states
    fbRunCallCtrl:          FB_InvocationControl;
END_VAR

METHOD AddState : BOOL
VAR_INPUT
    ipState:        I_State;
END_VAR
IF ipState = 0
    OR_ELSE THIS^.Contains(ipState) THEN
    RETURN;
END_IF

AddState := THIS^.fbStateList.AddItem(ipState) <> -1;
IF AddState THEN
    THIS^.TryAssignSelfToState(ipState);
END_IF
END_METHOD

METHOD ClearStates
VAR
    i:          DINT;
    ipState:    I_State;
END_VAR
FOR i := 0 TO THIS^.nLastIdx DO
    THIS^.TryMakeStateOrphan(THIS^.StateAt(i));
END_FOR

THIS^.fbStateList.Clear();
THIS^._ipPrevState := THIS^._ipState;
THIS^._ipState := 0;
END_METHOD

METHOD Contains : BOOL
VAR_INPUT
    ipState:        I_State;
END_VAR
Contains := THIS^.fbStateList.Contains(ipState);
END_METHOD

// Previous state
PROPERTY ipPrevState : I_State
GET
ipPrevState := THIS^._ipPrevState;
END_GET
END_PROPERTY

// Current state
PROPERTY ipState : I_State
GET
ipState := THIS^._ipState;
END_GET
END_PROPERTY

PROPERTY PROTECTED nLastIdx : DINT
GET
IF THIS^.fbStateList.nCount > 0 THEN
    nLastIdx := TO_DINT(THIS^.fbStateList.nCount - 1);
END_IF
END_GET
END_PROPERTY

PROPERTY nStateChangeCount : UDINT
GET
nStateChangeCount := THIS^._nStateChangeCount;
END_GET
END_PROPERTY

PROPERTY nStateCount : UDINT
GET
nStateCount := THIS^.fbStateList.nCount;
END_GET
END_PROPERTY

METHOD Restore : I_Restorable
VAR_INPUT
END_VAR
Restore := THIS^;
END_METHOD

METHOD Run
THIS^.fbRunCallCtrl.Track();

IF THIS^._ipState <> 0 THEN
    THIS^._ipState.Run();
ELSE
    IF THIS^.fbRunCallCtrl.bNewInvocation THEN
        Tc2_System.ADSLOGSTR(msgCtrlMask := Tc2_System.ADSLOG_MSGTYPE_ERROR,
                             msgFmtStr := 'Current state for %s is not yet initialized',
                             strArg := THIS^.sPath);
    END_IF
END_IF
END_METHOD

METHOD SetState : BOOL
VAR_INPUT
    newState:           I_State;
END_VAR
VAR_INST
    fbCallCtrl:         FB_InvocationControl;
END_VAR
fbCallCtrl.Track();

IF NOT THIS^.fbRunCallCtrl.bCalledCyclically THEN
    IF fbCallCtrl.bNewInvocation THEN
        Tc2_System.ADSLOGSTR(msgCtrlMask := Tc2_System.ADSLOG_MSGTYPE_ERROR,
                             msgFmtStr := '%s state machine is not being runned',
                             strArg := THIS^.sPath);
    END_IF
END_IF

IF newState = 0
    OR_ELSE newState = THIS^.ipState THEN
    RETURN;
END_IF

IF fbStateList.nCount <= 0 THEN
    IF fbCallCtrl.bNewInvocation THEN
        Tc2_System.ADSLOGSTR(msgCtrlMask := Tc2_System.ADSLOG_MSGTYPE_ERROR,
                             msgFmtStr := '%s state machine is empty, please add states to the state machine',
                             strArg := THIS^.sPath);
    END_IF

    RETURN;
END_IF

IF NOT THIS^.fbStateList.Contains(newState) THEN
    RETURN;
END_IF

IF THIS^._ipState <> 0 THEN
    THIS^._ipState.OnExit();
END_IF

THIS^._ipPrevState := _ipState;
THIS^._ipState := newState;

IF THIS^._ipState <> 0 THEN
    THIS^._ipState.OnEntry();
END_IF

THIS^._nStateChangeCount := THIS^._nStateChangeCount + 1;

SetState := TRUE;
END_METHOD

METHOD StateAt : I_State
VAR_INPUT
    nIdx:       DINT; // Zero-based index to list of state
END_VAR
VAR
    ipObject:   I_Object;
END_VAR
ipObject := THIS^.fbStateList.ItemAt(nIdx);

IF ipObject <> 0 THEN
    __QUERYINTERFACE(ipObject, StateAt);
END_IF
END_METHOD

METHOD PROTECTED TryAssignSelfToState : BOOL
VAR_INPUT
    ipState:        I_State;
END_VAR
IF ipState <> 0
    AND_THEN THIS^.fbStateList.Contains(ipState) THEN
    ipState.AssignStateMachine(THIS^);
    TryAssignSelfToState := TRUE;
END_IF
END_METHOD

METHOD PROTECTED TryMakeStateOrphan : BOOL
VAR_INPUT
    ipState:        I_State;
END_VAR
IF ipState <> 0 THEN
    ipState.MakeOrphan();
    TryMakeStateOrphan := TRUE;
END_IF
END_METHOD

END_FUNCTION_BLOCK

// ---- State Pattern/Tests/Test Subjects/FB_State1.TcPOU
FUNCTION_BLOCK INTERNAL FB_State1 EXTENDS FB_State
VAR_INPUT
END_VAR
VAR_OUTPUT
END_VAR
VAR
END_VAR

END_FUNCTION_BLOCK

// ---- State Pattern/FB_State.TcPOU
FUNCTION_BLOCK ABSTRACT FB_State EXTENDS FB_Object IMPLEMENTS I_State
VAR
    _ipStateMachine:        I_StateMachine;
END_VAR

METHOD AssignStateMachine : BOOL
VAR_INPUT
    ipStateMachine:     I_StateMachine;
END_VAR
IF ipStateMachine <> 0
    AND_THEN THIS^._ipStateMachine = 0 THEN
    THIS^._ipStateMachine := ipStateMachine;
    AssignStateMachine := TRUE;
END_IF
END_METHOD

METHOD FB_init : BOOL
VAR_INPUT
    bInitRetains:           BOOL; // if TRUE, the retain variables are initialized (warm start / cold start)
    bInCopyCode:            BOOL;  // if TRUE, the instance afterwards gets moved into the copy code (online change)
    ipStateMachine:         I_StateMachine;
END_VAR
IF ipStateMachine <> 0 THEN
    ipStateMachine.AddState(THIS^);
END_IF
END_METHOD

PROPERTY ipStateMachine : I_StateMachine
GET
ipStateMachine := THIS^._ipStateMachine;
END_GET
END_PROPERTY

METHOD MakeOrphan
VAR_INPUT
END_VAR
THIS^._ipStateMachine := 0;
END_METHOD

METHOD OnEntry
VAR_INPUT
END_VAR
END_METHOD

METHOD OnExit
VAR_INPUT
END_VAR
END_METHOD

METHOD Restore : I_Restorable
VAR_INPUT
END_VAR
Restore := THIS^;
END_METHOD

METHOD Run
VAR_INPUT
END_VAR
END_METHOD

END_FUNCTION_BLOCK

// ---- State Pattern/Tests/Test Subjects/FB_State2.TcPOU
FUNCTION_BLOCK INTERNAL FB_State2 EXTENDS FB_State
VAR_INPUT
END_VAR
VAR_OUTPUT
END_VAR
VAR
END_VAR

END_FUNCTION_BLOCK

// ---- State Pattern/Tests/Test Subjects/FB_State3.TcPOU
FUNCTION_BLOCK INTERNAL FB_State3 EXTENDS FB_State
VAR_INPUT
END_VAR
VAR_OUTPUT
END_VAR
VAR
END_VAR

END_FUNCTION_BLOCK

// ---- State Pattern/Tests/Test Subjects/FB_State4.TcPOU
FUNCTION_BLOCK INTERNAL FB_State4 EXTENDS FB_State
VAR_INPUT
END_VAR
VAR_OUTPUT
END_VAR
VAR
END_VAR

END_FUNCTION_BLOCK

// ---- State Pattern/Tests/Test Subjects/FB_Year.TcPOU
FUNCTION_BLOCK INTERNAL FB_Year EXTENDS FB_Object IMPLEMENTS I_SeasonControl, I_CyclicTask
VAR
    fbSeasonStateMachine:   FB_SeasonStateMachine;
    fbWinter:               FB_Winter(THIS^.fbSeasonStateMachine, THIS^);
    fbSpring:               FB_Spring(THIS^.fbSeasonStateMachine, THIS^);
    fbSummer:               FB_Summer(THIS^.fbSeasonStateMachine, THIS^);
    fbAutumn:               FB_Autumn(THIS^.fbSeasonStateMachine, THIS^);

    nCounter:               UDINT;
    nModVal:                UDINT := 500;
END_VAR

METHOD ChangeToSummerTyres
VAR_INPUT
END_VAR
THIS^.CurrentState().ChangeToSummerTyres();
END_METHOD

METHOD ChangeToWinterTyres
VAR_INPUT
END_VAR
THIS^.CurrentState().ChangeToWinterTyres();
END_METHOD

METHOD CurrentState : I_SeasonState
__QUERYINTERFACE(THIS^.fbSeasonStateMachine.ipState, CurrentState);
END_METHOD

METHOD FB_init : BOOL
VAR_INPUT
    bInitRetains:           BOOL; // if TRUE, the retain variables are initialized (warm start / cold start)
    bInCopyCode:            BOOL;  // if TRUE, the instance afterwards gets moved into the copy code (online change)
END_VAR
THIS^.fbSeasonStateMachine.SetState(THIS^.StateSummer);
THIS^.CurrentState().ChangeToSummerTyres();
END_METHOD

METHOD NextSeason
VAR_INPUT
END_VAR
THIS^.fbSeasonStateMachine.NextSeason();
END_METHOD

METHOD Run
VAR_INPUT
END_VAR
THIS^.nCounter := THIS^.nCounter + 1;
THIS^.fbSeasonStateMachine.Run();
END_METHOD

PROPERTY StateAutumn : I_State
GET
StateAutumn := THIS^.fbAutumn;
END_GET
END_PROPERTY

PROPERTY StateSpring : I_State
GET
StateSpring := THIS^.fbSpring;
END_GET
END_PROPERTY

PROPERTY StateSummer : I_State
GET
StateSummer := THIS^.fbSummer;
END_GET
END_PROPERTY

PROPERTY StateWinter : I_State
GET
StateWinter := THIS^.fbWinter;
END_GET
END_PROPERTY

END_FUNCTION_BLOCK

// ---- State Pattern/Tests/Test Subjects/FB_SeasonStateMachine.TcPOU
FUNCTION_BLOCK INTERNAL FB_SeasonStateMachine EXTENDS FB_StateMachine
VAR
    fbDefaultState:     FB_Default(THIS^, THIS^);
END_VAR

METHOD CurrentSeason : I_SeasonState
VAR_INPUT
END_VAR
__QUERYINTERFACE(THIS^.ipState, CurrentSeason);

IF CurrentSeason = 0 THEN
    CurrentSeason := THIS^.fbDefaultState;
END_IF
END_METHOD

METHOD NextSeason
VAR_INPUT
END_VAR
THIS^.CurrentSeason().NextSeason();
END_METHOD

PROPERTY StateDefault : I_SeasonState
GET
StateDefault := THIS^.fbDefaultState;
END_GET
END_PROPERTY

END_FUNCTION_BLOCK

// ---- State Pattern/Tests/Test Subjects/FB_Default.TcPOU
FUNCTION_BLOCK INTERNAL FB_Default EXTENDS FB_SeasonBase
VAR
END_VAR

METHOD  NextSeason
VAR_INST
    fbCallCtrl:     FB_InvocationControl;
END_VAR
IF fbCallCtrl.Track().bNewInvocation THEN
    Tc2_System.ADSLOGSTR(msgCtrlMask := THIS^._nLogLevel,
                         msgFmtStr := 'Current state for %s is not initialized!',
                         strArg := THIS^.sPath);
END_IF

IF THIS^.ipStateMachine <> 0 THEN
    THIS^.ipStateMachine.SetState(THIS^);
END_IF
END_METHOD

END_FUNCTION_BLOCK

// ---- State Pattern/Tests/Test Subjects/FB_SeasonBase.TcPOU
FUNCTION_BLOCK INTERNAL ABSTRACT FB_SeasonBase EXTENDS FB_State IMPLEMENTS I_SeasonState
VAR
    _ipWeatherCtrl:     I_SeasonControl;
    _eState:            E_Season;
END_VAR
VAR_STAT
    _bWindBlowing:      BOOL;
    _bRaining:          BOOL;
    _bSunShining:       BOOL;
    _bSnowing:          BOOL;
    _nTyresType:        BYTE; // 0: winter, 1: summer/all season
    _nLeavesState:      BYTE; // 0: no leave, 1: green leaves, 2: yellow/orange/red leaves
    _nCounter:          UDINT;
    _nModVal:           UDINT := 500;
    _nLogLevel:         DWORD := Tc2_System.ADSLOG_MSGTYPE_WARN;
END_VAR

PROPERTY FINAL bRaining : BOOL
GET
bRaining := THIS^._bRaining;
END_GET
END_PROPERTY

PROPERTY FINAL bSnowing : BOOL
GET
bSnowing := THIS^._bSnowing;
END_GET
END_PROPERTY

PROPERTY FINAL bSunShining : BOOL
GET
bSunShining := THIS^._bSunShining;
END_GET
END_PROPERTY

PROPERTY FINAL bWindBlowing : BOOL
GET
bWindBlowing := THIS^._bWindBlowing;
END_GET
END_PROPERTY

METHOD ChangeToSummerTyres
VAR_INPUT
END_VAR
END_METHOD

METHOD ChangeToWinterTyres
VAR_INPUT
END_VAR
END_METHOD

PROPERTY FINAL eState : E_Season
GET
eState := THIS^._eState;
END_GET
END_PROPERTY

METHOD FB_init : BOOL
VAR_INPUT
    bInitRetains:           BOOL; // if TRUE, the retain variables are initialized (warm start / cold start)
    bInCopyCode:            BOOL;  // if TRUE, the instance afterwards gets moved into the copy code (online change)
    ipStateMachine:         I_StateMachine;
    ipParentObject:         I_Object;
END_VAR
__QUERYINTERFACE(ipParentObject, THIS^._ipWeatherCtrl);
END_METHOD

PROPERTY ipSeasonCtrl : I_SeasonControl
GET
ipSeasonCtrl := THIS^._ipWeatherCtrl;
END_GET
END_PROPERTY

METHOD ABSTRACT NextSeason
VAR_INPUT
END_VAR
END_METHOD

PROPERTY FINAL nLeavesState : BYTE
GET
nLeavesState := THIS^._nLeavesState;
END_GET
END_PROPERTY

PROPERTY FINAL nTyresType : BYTE
GET
nTyresType := THIS^._nTyresType;
END_GET
END_PROPERTY

METHOD OnEntry
VAR
    sTmp:       STRING(MAX_STRING_LENGTH);
END_VAR
sTmp := CONCAT(THIS^.sState, ' here we go!');

Tc2_System.ADSLOGSTR(msgCtrlMask := THIS^._nLogLevel,
                     msgFmtStr := sTmp,
                     strArg := '');

IF THIS^.bWindBlowing THEN
    Tc2_System.ADSLOGSTR(msgCtrlMask := THIS^._nLogLevel,
                         msgFmtStr := 'The wind is blowing',
                         strArg := '');
END_IF

IF THIS^.bRaining THEN
    Tc2_System.ADSLOGSTR(msgCtrlMask := THIS^._nLogLevel,
                         msgFmtStr := 'It$'s raining dogs and cats',
                         strArg := '');
END_IF

IF THIS^.bSunShining THEN
    Tc2_System.ADSLOGSTR(msgCtrlMask := THIS^._nLogLevel,
                         msgFmtStr := 'Aurinko paistaa',
                         strArg := '');
END_IF

IF THIS^.bSnowing THEN
    Tc2_System.ADSLOGSTR(msgCtrlMask := THIS^._nLogLevel,
                         msgFmtStr := 'Sataa lunta',
                         strArg := '');
END_IF
END_METHOD

METHOD OnExit
VAR
    sTmp:       STRING(MAX_STRING_LENGTH);
END_VAR
sTmp := CONCAT('Good bye ', THIS^.sState);

Tc2_System.ADSLOGSTR(msgCtrlMask := THIS^._nLogLevel,
                     msgFmtStr := sTmp,
                     strArg := '');
END_METHOD

METHOD Run
VAR_INPUT
END_VAR
THIS^._nCounter := THIS^._nCounter + 1;
END_METHOD

PROPERTY FINAL sState : STRING(MAX_STRING_LENGTH)
GET
sState := TO_STRING(THIS^.eState);
END_GET
END_PROPERTY

END_FUNCTION_BLOCK

// ---- State Pattern/Tests/Test Subjects/FB_Winter.TcPOU
FUNCTION_BLOCK INTERNAL FB_Winter EXTENDS FB_SeasonBase
VAR
END_VAR

METHOD ChangeToWinterTyres
VAR_INPUT
END_VAR
THIS^._nTyresType := 0;
Tc2_System.ADSLOGSTR(msgCtrlMask := THIS^._nLogLevel,
                     msgFmtStr := 'Changed to winter tyres',
                     strArg := '');
END_METHOD

METHOD FB_init : BOOL
VAR_INPUT
    bInitRetains:           BOOL; // if TRUE, the retain variables are initialized (warm start / cold start)
    bInCopyCode:            BOOL;  // if TRUE, the instance afterwards gets moved into the copy code (online change)
    ipStateMachine:         I_StateMachine;
    ipParentObject:         I_Object;
END_VAR
THIS^._eState := E_Season.Winter;
END_METHOD

METHOD  NextSeason
VAR_INPUT
END_VAR
THIS^.ipStateMachine.SetState(THIS^.ipSeasonCtrl.StateSpring);
END_METHOD

METHOD OnEntry
VAR_INPUT
END_VAR
SUPER^.OnEntry();
THIS^._bWindBlowing     := FALSE;
THIS^._bRaining         := FALSE;
THIS^._bSunShining      := FALSE;
THIS^._bSnowing         := TRUE;
THIS^._nLeavesState     := 0;
END_METHOD

END_FUNCTION_BLOCK

// ---- State Pattern/Tests/Test Subjects/FB_Spring.TcPOU
FUNCTION_BLOCK INTERNAL FB_Spring EXTENDS FB_SeasonBase
VAR_INPUT
END_VAR
VAR_OUTPUT
END_VAR
VAR
END_VAR

METHOD ChangeToSummerTyres
VAR_INPUT
END_VAR
THIS^._nTyresType := 1;
Tc2_System.ADSLOGSTR(msgCtrlMask := THIS^._nLogLevel,
                     msgFmtStr := 'Changed to summer tyres',
                     strArg := '');
END_METHOD

METHOD FB_init : BOOL
VAR_INPUT
    bInitRetains:           BOOL; // if TRUE, the retain variables are initialized (warm start / cold start)
    bInCopyCode:            BOOL;  // if TRUE, the instance afterwards gets moved into the copy code (online change)
    ipStateMachine:         I_StateMachine;
    ipParentObject:         I_Object;
END_VAR
THIS^._eState := E_Season.Spring;
END_METHOD

METHOD  NextSeason
VAR_INPUT
END_VAR
THIS^.ipStateMachine.SetState(THIS^.ipSeasonCtrl.StateSummer);
END_METHOD

METHOD OnEntry
VAR_INPUT
END_VAR
SUPER^.OnEntry();
THIS^._bWindBlowing     := FALSE;
THIS^._bRaining         := TRUE;
THIS^._bSunShining      := FALSE;
THIS^._bSnowing         := TRUE;
THIS^._nLeavesState     := 1;
END_METHOD

METHOD OnExit
SUPER^.OnExit();
THIS^._bWindBlowing     := FALSE;
THIS^._bRaining         := FALSE;
THIS^._bSunShining      := FALSE;
THIS^._bSnowing         := TRUE;
THIS^._nLeavesState     := 1;
END_METHOD

END_FUNCTION_BLOCK

// ---- State Pattern/Tests/Test Subjects/FB_Summer.TcPOU
FUNCTION_BLOCK INTERNAL FB_Summer EXTENDS FB_SeasonBase
VAR_INPUT
END_VAR
VAR_OUTPUT
END_VAR
VAR
END_VAR

METHOD ChangeToSummerTyres
VAR_INPUT
END_VAR
THIS^._nTyresType := 1;
Tc2_System.ADSLOGSTR(msgCtrlMask := THIS^._nLogLevel,
                     msgFmtStr := 'Changed to summer tyres',
                     strArg := '');
END_METHOD

METHOD FB_init : BOOL
VAR_INPUT
    bInitRetains:           BOOL; // if TRUE, the retain variables are initialized (warm start / cold start)
    bInCopyCode:            BOOL;  // if TRUE, the instance afterwards gets moved into the copy code (online change)
    ipStateMachine:         I_StateMachine;
    ipParentObject:         I_Object;
END_VAR
THIS^._eState := E_Season.Summer;
END_METHOD

METHOD  NextSeason
VAR_INPUT
END_VAR
THIS^.ipStateMachine.SetState(THIS^.ipSeasonCtrl.StateAutumn);
END_METHOD

METHOD OnEntry
SUPER^.OnEntry();
THIS^._bWindBlowing     := FALSE;
THIS^._bRaining         := FALSE;
THIS^._bSunShining      := TRUE;
THIS^._bSnowing         := FALSE;
THIS^._nLeavesState     := 1;
END_METHOD

END_FUNCTION_BLOCK

// ---- State Pattern/Tests/Test Subjects/FB_Autumn.TcPOU
FUNCTION_BLOCK INTERNAL FB_Autumn EXTENDS FB_SeasonBase
VAR_INPUT
END_VAR
VAR_OUTPUT
END_VAR
VAR
END_VAR

METHOD FB_init : BOOL
VAR_INPUT
    bInitRetains:           BOOL; // if TRUE, the retain variables are initialized (warm start / cold start)
    bInCopyCode:            BOOL;  // if TRUE, the instance afterwards gets moved into the copy code (online change)
    ipStateMachine:         I_StateMachine;
    ipParentObject:         I_Object;
END_VAR
THIS^._eState := E_Season.Autumn;
END_METHOD

METHOD  NextSeason
VAR_INPUT
END_VAR
THIS^.ipStateMachine.SetState(THIS^.ipSeasonCtrl.StateWinter);
END_METHOD

METHOD OnEntry
VAR_INPUT
END_VAR
SUPER^.OnEntry();
THIS^._bWindBlowing     := TRUE;
THIS^._bRaining         := FALSE;
THIS^._bSunShining      := FALSE;
THIS^._bSnowing         := FALSE;
THIS^._nLeavesState     := 2;

Tc2_System.ADSLOGSTR(msgCtrlMask := THIS^._nLogLevel,
                     msgFmtStr := 'Leaves are changing color to yellow/orange/bright red',
                     strArg := '');
END_METHOD

METHOD OnExit
SUPER^.OnExit();
THIS^._bWindBlowing     := FALSE;
THIS^._bRaining         := FALSE;
THIS^._bSunShining      := FALSE;
THIS^._bSnowing         := FALSE;
THIS^._nLeavesState     := 2;
END_METHOD

END_FUNCTION_BLOCK

// ---- Action/Tests/FB_Action_Test.TcPOU
FUNCTION_BLOCK INTERNAL FB_Action_Test EXTENDS TcUnit.FB_TestSuite
VAR
END_VAR

TestActivateAction();
TestRunCyclicTaskAction();

METHOD PRIVATE TestActivateAction
VAR_INST
    fbObject: FB_ActionTestObject;
    fbActivate: FB_ActivateAction;
END_VAR
TcUnit.TEST('TestActivateTaskAction');

THIS^.AssertFalse(Condition := fbObject.bIsActivated,
                  Message := 'Object should not be activated yet');

fbActivate.Inputs(TRUE).Execute(fbObject);

THIS^.AssertTrue(Condition := fbObject.bIsActivated,
                 Message := 'Failed to activate object');

fbActivate.Inputs(FALSE).Execute(fbObject);

THIS^.AssertFalse(Condition := fbObject.bIsActivated,
                  Message := 'Failed to deactivate object');

TcUnit.TEST_FINISHED();
END_METHOD

METHOD PRIVATE TestRunCyclicTaskAction
VAR_INST
    nCyclesToRun: UDINT := 5;
    nCounter: UDINT := 0;
    fbObject: FB_ActionTestObject;
    fbRunCyclicTask: FB_RunCyclicTasksAction;
END_VAR
TcUnit.TEST('TestRunCyclicTaskAction');

fbRunCyclicTask.Execute(fbObject);
nCounter := nCounter + 1;

IF nCyclesToRun = nCounter THEN
    THIS^.AssertEquals_UDINT(Expected := nCyclesToRun,
                             Actual := fbObject.nCounter,
                             Message := 'Unexpected counter value of cyclic object');
    TcUnit.TEST_FINISHED();
END_IF
END_METHOD

END_FUNCTION_BLOCK

// ---- Context/FB_Context.TcPOU
{attribute 'reflection'}
FUNCTION_BLOCK ABSTRACT FB_Context IMPLEMENTS I_Context, I_CyclicTask
VAR
    _nIdentity:         ULINT;
    _ipSelf:            I_Object;

    {attribute 'instance-path'}
    {attribute 'noinit'}
    _sPath:             STRING(MAX_STRING_LENGTH);
END_VAR

METHOD Equals : BOOL
VAR_INPUT
    ipObject:       I_Object;
END_VAR
Equals := ipObject = THIS^._ipSelf;
END_METHOD

METHOD FB_init : BOOL
VAR_INPUT
	bInitRetains : BOOL; // if TRUE, the retain variables are initialized (warm start / cold start)
	bInCopyCode : BOOL;  // if TRUE, the instance afterwards gets moved into the copy code (online change)
END_VAR
THIS^._nIdentity := ADR(THIS^);
THIS^._ipSelf := THIS^;
END_METHOD

PROPERTY ipContext : I_Context
GET
ipContext := THIS^;
END_GET
END_PROPERTY

METHOD PROTECTED ABSTRACT Main
VAR_INPUT
END_VAR
END_METHOD

PROPERTY nIdentity : ULINT
GET
nIdentity := ADR(THIS^);
END_GET
END_PROPERTY

METHOD PROTECTED OnEntry
VAR_INPUT
END_VAR
END_METHOD

METHOD PROTECTED OnExit
VAR_INPUT
END_VAR
END_METHOD

METHOD FINAL Run
VAR_INPUT
END_VAR
THIS^.OnEntry();
THIS^.Main();
THIS^.OnExit();
END_METHOD

PROPERTY sPath : STRING(MAX_STRING_LENGTH)
GET
sPath := THIS^._sPath;
END_GET
END_PROPERTY

END_FUNCTION_BLOCK

// ---- Object/FB_LinkedObject.TcPOU
FUNCTION_BLOCK ABSTRACT FB_LinkedObject EXTENDS FB_Object IMPLEMENTS I_Object
VAR
    _ipParent:          I_LinkedObject;
END_VAR

METHOD FB_init : BOOL
VAR_INPUT
    bInitRetains:           BOOL; // if TRUE, the retain variables are initialized (warm start / cold start)
    bInCopyCode:            BOOL;  // if TRUE, the instance afterwards gets moved into the copy code (online change)
    ipParentObject:         I_LinkedObject;
END_VAR
THIS^._ipParent := ipParentObject;
END_METHOD

PROPERTY ipContext : I_Context
GET
IF THIS^._ipParent <> 0 THEN
    ipContext := THIS^.ipParent.ipContext;
END_IF
END_GET
END_PROPERTY

PROPERTY ipParent : I_LinkedObject
GET
ipParent := THIS^._ipParent;
END_GET
END_PROPERTY

END_FUNCTION_BLOCK
